FUNCTION toErrorEventArray : ARRAY [0..5] OF ST_Event
VAR_INPUT
	errorEvents 	: ST_ErrorEvents;    
END_VAR
VAR
	arrEvents 		: ARRAY [0..5] OF ST_Event;
END_VAR

arrEvents[0] := errorEvents.PressureDiffEvaporatorTooHigh;
arrEvents[1] := errorEvents.LowPressureRefrigerationThermostat;
arrEvents[2] := errorEvents.HighPressureRefrigerationThermostat;
arrEvents[3] := errorEvents.MotorProtectionTriggered;
arrEvents[4] := errorEvents.ExpansionValveTriggered;

ToErrorEventArray := arrEvents;

END_FUNCTION

(* stored: Version 1.1.0.1
   POU toErrorEventArray: Id {dfa38065-b5cf-4a1b-bb0e-be59257fcadc}, SpecialFunc None *)
